FUNCTION_BLOCK BfbWaterPump
  (* Standard: 61499-2 *)
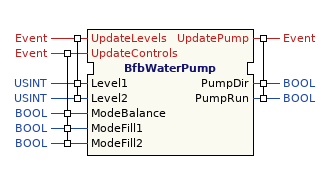
  EVENT_INPUT
    UpdateLevels WITH Level1, Level2;
    UpdateControls WITH ModeBalance, ModeFill1, ModeFill2;
  END_EVENT
  EVENT_OUTPUT
    UpdatePump WITH PumpDir, PumpRun;
  END_EVENT
  VAR_INPUT
    Level1 : USINT := 0;
    Level2 : USINT := 0;
    ModeBalance : BOOL;
    ModeFill1 : BOOL;
    ModeFill2 : BOOL;
  END_VAR
  VAR_OUTPUT
    PumpDir : BOOL := 0;
    PumpRun : BOOL := 0;
  END_VAR
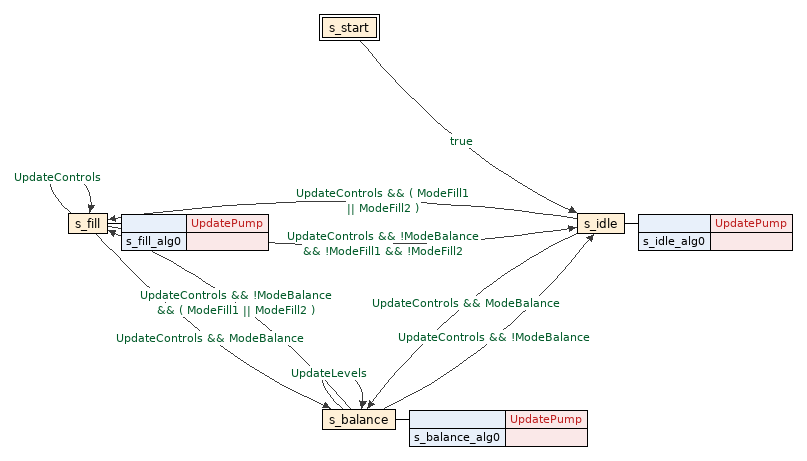
  EC_STATES
    s_start;
    s_idle : -> UpdatePump, s_idle_alg0;
    s_balance : -> UpdatePump, s_balance_alg0;
    s_fill : -> UpdatePump, s_fill_alg0;
  END_STATES
  EC_TRANSITIONS
    s_start TO s_idle := true;
    s_idle TO s_balance := UpdateControls && ModeBalance;
    s_idle TO s_fill := UpdateControls && ( ModeFill1 || ModeFill2 );
    s_balance TO s_fill := UpdateControls && !ModeBalance && ( ModeFill1 || ModeFill2 );
    s_balance TO s_idle := UpdateControls && !ModeBalance;
    s_balance TO s_balance := UpdateLevels;
    s_fill TO s_balance := UpdateControls && ModeBalance;
    s_fill TO s_idle := UpdateControls && !ModeBalance && !ModeFill1 && !ModeFill2;
    s_fill TO s_fill := UpdateControls;
  END_TRANSITIONS
  ALGORITHM s_idle_alg0 IN ST:
PumpDir := 0; PumpRun := 0;
  END_ALGORITHM
  ALGORITHM s_balance_alg0 IN ST:
                if Level1 > Level2 then
                    PumpDir := 0;
                    PumpRun := 1;
                elsif Level2 > Level1 then
                    PumpDir := 1;
                    PumpRun := 1;
                else
                    PumpRun := 0;
                end_if;
  END_ALGORITHM
  ALGORITHM s_fill_alg0 IN ST:
                if ModeFill1 then
                    PumpDir := 1;
                    PumpRun := 1;
                elsif ModeFill2 then
                    PumpDir := 0;
                    PumpRun := 1;
                else
                    PumpRun := 0;
                end_if;
  END_ALGORITHM
END_FUNCTION_BLOCK
